INTERFACE I_EquipmentModule_SR EXTENDS I_PackML_BaseModule

PROPERTY EquipmentModuleID : E_EM_Index;
GET
END_GET
SET
END_SET
END_PROPERTY

PROPERTY InSimulation : BOOL
SET
END_SET
END_PROPERTY

PROPERTY SafetyOK : BOOL
SET
END_SET
END_PROPERTY

METHOD SimulationOff : BOOL
VAR_INPUT
END_VAR
END_METHOD

METHOD SimulationOn : BOOL
VAR_INPUT
END_VAR
END_METHOD

END_INTERFACE

(* stored: Version 1.1.0.1
   Itf I_EquipmentModule_SR: Id {d663814b-0dd5-4c05-8ee9-d9773ef737eb}
   Property EquipmentModuleID: Id {aeff10e9-5bc3-42e0-bd24-7b6a3103bb95}
   Get Get: Id {f734c3d3-2b44-410a-88d3-1b60e7d95c75}
   Set Set: Id {0d1cab90-1e3c-4164-9234-459c105cd813}
   Property InSimulation: Id {ff9c8eaf-dfa5-416b-b4c5-c6ed5a3e6add}
   Set Set: Id {291cfa6e-3fd2-41f2-9fe7-a70cb02d95ba}
   Property SafetyOK: Id {566ec046-912c-42db-96cc-8cfb6cddf5c7}
   Set Set: Id {966bba5b-9b8b-40ab-8c92-e5e90b0d7d0b}
   Method SimulationOff: Id {3e2deaa5-a795-4d7d-a053-15eee544bf9c}
   Method SimulationOn: Id {bb03762e-6c33-4760-9d9f-bc19309e2d8f} *)
